// Mitsubishi GX Works2 project: PLC_GROUP_1   PLC: FX3G

// global labels: Global1
VAR_GLOBAL
  Start_day AT X007 : BOOL;
  Emergency_button AT X005 : BOOL;
  Inventory_check_flag AT M12 : BOOL;
  Day_activation_flag AT M0 : BOOL;
  Active_day AT Y007 : BOOL;
  Valid_inventory_flag AT M10 : BOOL;
  Start_making_flag AT M11 : BOOL;
  Special_gumigum_making AT M2 : BOOL;
  Regular_gumigum_making AT M1 : BOOL;
  Inventory_check AT X001 : BOOL;
  Petel_invetory AT D1200 : INT;
  Lemon_invetory AT D1202 : INT;
  Staiblaizer_invetory AT D1204 : INT;
  Gummy_bear_invetory AT D1206 : INT;
  Lemon AT D1112 : INT;
  Staibliazer AT D1114 : INT;
  Gummy_bear AT D1116 : INT;
  Analog_input AT D8280 : INT;
  IC_making_timer AT TC0 : BOOL;
  IC_making_timer_aprv AT TS0 : BOOL;
  Freezing_Timer AT TC1 : BOOL;
  Freezing_Timer_Aprv AT TS1 : BOOL;
  Regular_gumigum_mixing AT TC2 : BOOL;
  Regular_gumigum_mixing_apv AT TS2 : BOOL;
  Special_gumigum_mixing AT TC3 : BOOL;
  Special_gumigum_mixing_apv AT TS3 : BOOL;
  Flashlight_timer1 AT TC4 : BOOL;
  Flashlight_timer1_apv AT TS4 : BOOL;
  Flashlight_timer2 AT TC5 : BOOL;
  Flashlight_timer2_apv AT TS5 : BOOL;
  Start_mixing AT M13 : BOOL;
END_VAR
VAR_GLOBAL CONSTANT
  Constant2000 : INT := 2000;
  Constant2400 : INT := 2400;
  Req_petel_reg : INT := 280;
  Req_lemon_reg : INT := 455;
  Req_staibelaizer_reg : INT := 105;
  Req_gummybear_reg : INT := 28;
  Req_petel_spec : INT := 385;
  Req_lemon_spec : INT := 665;
  Req_staibelaizer_spec : INT := 210;
  Req_gummybear_spec : INT := 70;
END_VAR
VAR_GLOBAL
  Petel AT D1110 : INT;
END_VAR
VAR_GLOBAL CONSTANT
  timer50 : INT := 50;
END_VAR
VAR_GLOBAL
  timerTc2 AT TC2 : BOOL;
  IC_making AT Y000 : BOOL;
  Freezing_button AT X002 : BOOL;
  Freezing_lamp AT Y002 : BOOL;
END_VAR
VAR_GLOBAL CONSTANT
  timer30 : INT := 30;
END_VAR
VAR_GLOBAL
  Invalid_analog_input AT M14 : BOOL;
END_VAR
VAR_GLOBAL CONSTANT
  Regular_petel_container : INT := 350;
  Regular_lemon_container : INT := 490;
  Special_petel_container : INT := 560;
  Special_lemon_container : INT := 700;
END_VAR
VAR_GLOBAL
  Container_petel_IC AT D1130 : INT;
  Container_lemon_IC AT D1132 : INT;
  Petel_freezing_container AT D1140 : INT;
  Lemon_freezing_container AT D1142 : INT;
  Start_Freezing_Flag AT M15 : BOOL;
END_VAR
VAR_GLOBAL CONSTANT
  timer80 : INT := 80;
END_VAR
VAR_GLOBAL
  Temp_Sensor AT X003 : BOOL;
  Mixing_petel_container AT D1150 : INT;
  Mixing_lemon_container AT D1152 : INT;
  Flashlight_flag AT M16 : BOOL;
END_VAR
VAR_GLOBAL CONSTANT
  timer5 : INT := 5;
END_VAR
VAR_GLOBAL
  Flashlight1 AT Y005 : BOOL;
  Flashlight2 AT Y006 : BOOL;
  Packeges_counter AT D1160 : INT;
END_VAR
VAR_GLOBAL CONSTANT
  add1 : INT := 40;
END_VAR
VAR_GLOBAL
  Iteration_setting AT M30 : BOOL;
END_VAR
VAR_GLOBAL CONSTANT
  setting : INT;
END_VAR
VAR_GLOBAL
  Valid_p AT M40 : BOOL;
  Valid_l AT M41 : BOOL;
  Valid_s AT M42 : BOOL;
  Valid_g AT M43 : BOOL;
  check1 AT M50 : BOOL;
  check2 AT M51 : BOOL;
END_VAR
VAR_GLOBAL CONSTANT
  regular_gum : INT := 28;
  special_gum : INT := 70;
END_VAR
VAR_GLOBAL
  check3 AT M52 : BOOL;
  check4 AT M53 : BOOL;
  Analog_Output AT D8282 : INT;
END_VAR

// task Task_01 (event TRUE, interval 0, priority 31): POU_01

PROGRAM POU_01
(* structured ladder/FBD written out as ST: instructions are called as NAME(EN, inputs, outputs); _pN, _eN, _tN stand for wires *)
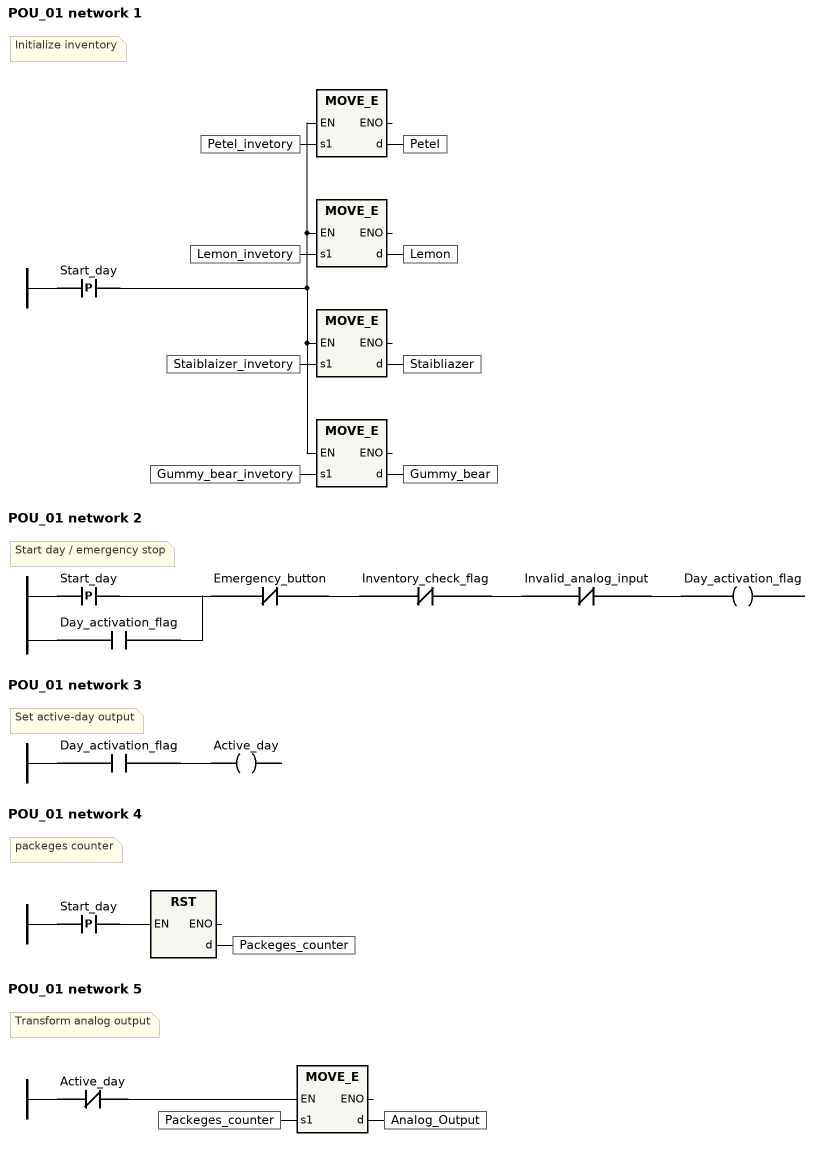
(* network 1 *)
(* Initialize inventory *)
_p1 := LDP(TRUE, Start_day);
MOVE_E(_p1, Petel_invetory, Petel);
MOVE_E(_p1, Lemon_invetory, Lemon);
MOVE_E(_p1, Staiblaizer_invetory, Staibliazer);
MOVE_E(_p1, Gummy_bear_invetory, Gummy_bear);
(* network 2 *)
(* Start day / emergency stop *)
Day_activation_flag := (((LDP(TRUE, Start_day) OR Day_activation_flag) AND NOT Emergency_button) AND NOT Inventory_check_flag) AND NOT Invalid_analog_input;
(* network 3 *)
(* Set active-day output *)
Active_day := Day_activation_flag;
(* network 4 *)
(* packeges counter *)
RST(LDP(TRUE, Start_day), Packeges_counter);
(* network 5 *)
(* Transform analog output *)
MOVE_E(NOT Active_day, Packeges_counter, Analog_Output);
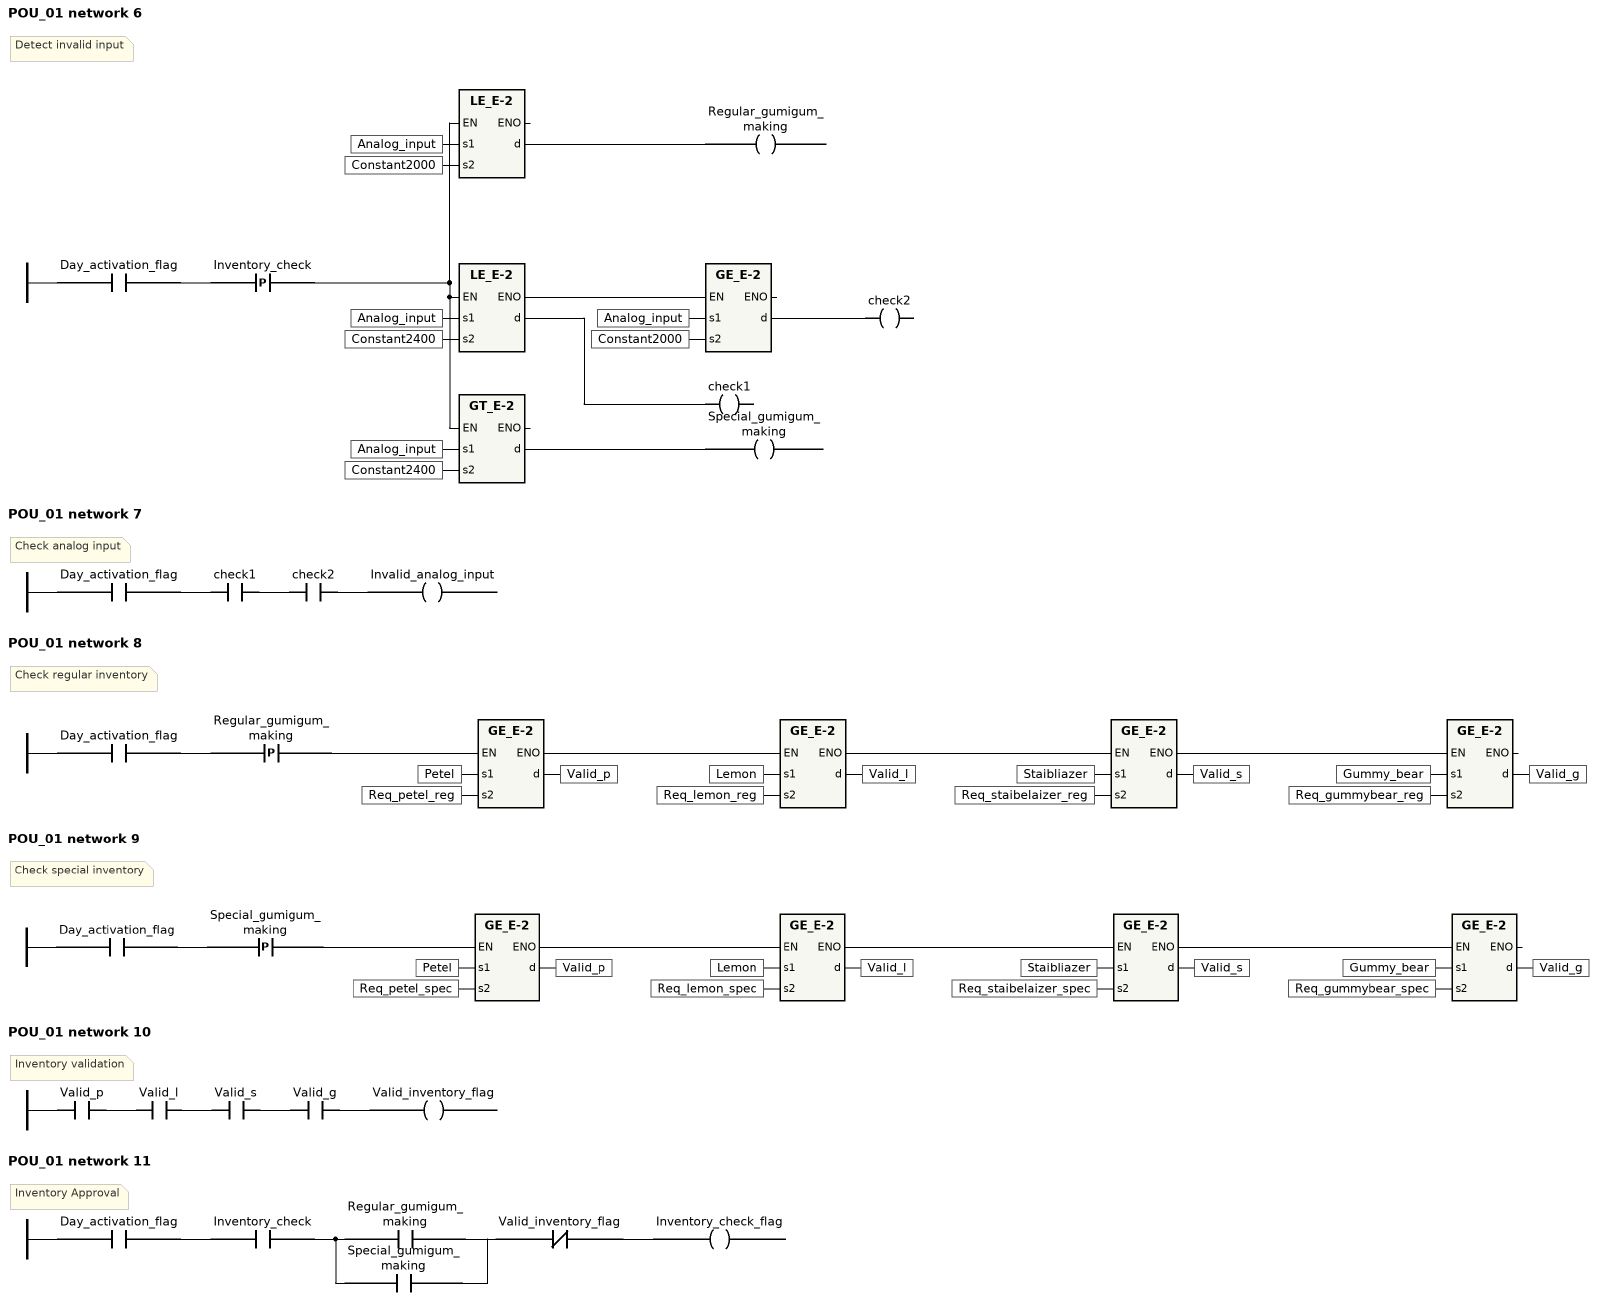
(* network 6 *)
(* Detect invalid input *)
_p1 := Day_activation_flag AND LDP(TRUE, Inventory_check);
LE_E(_p1, Analog_input, Constant2000, _t2);
Regular_gumigum_making := _t2;
GT_E(_p1, Analog_input, Constant2400, _t3);
Special_gumigum_making := _t3;
_e5 := LE_E(_p1, Analog_input, Constant2400, _t4);
GE_E(_e5, Analog_input, Constant2000, _t6);
check2 := _t6;
check1 := _t4;
(* network 7 *)
(* Check analog input *)
Invalid_analog_input := Day_activation_flag AND check1 AND check2;
(* network 8 *)
(* Check regular inventory *)
_e1 := GE_E(Day_activation_flag AND LDP(TRUE, Regular_gumigum_making), Petel, Req_petel_reg, Valid_p);
_e2 := GE_E(_e1, Lemon, Req_lemon_reg, Valid_l);
_e3 := GE_E(_e2, Staibliazer, Req_staibelaizer_reg, Valid_s);
GE_E(_e3, Gummy_bear, Req_gummybear_reg, Valid_g);
(* network 9 *)
(* Check special inventory *)
_e1 := GE_E(Day_activation_flag AND LDP(TRUE, Special_gumigum_making), Petel, Req_petel_spec, Valid_p);
_e2 := GE_E(_e1, Lemon, Req_lemon_spec, Valid_l);
_e3 := GE_E(_e2, Staibliazer, Req_staibelaizer_spec, Valid_s);
GE_E(_e3, Gummy_bear, Req_gummybear_spec, Valid_g);
(* network 10 *)
(* Inventory validation *)
Valid_inventory_flag := Valid_p AND Valid_l AND Valid_s AND Valid_g;
(* network 11 *)
(* Inventory Approval *)
_p1 := Day_activation_flag AND Inventory_check;
Inventory_check_flag := ((_p1 AND Regular_gumigum_making) OR (_p1 AND Special_gumigum_making)) AND NOT Valid_inventory_flag;
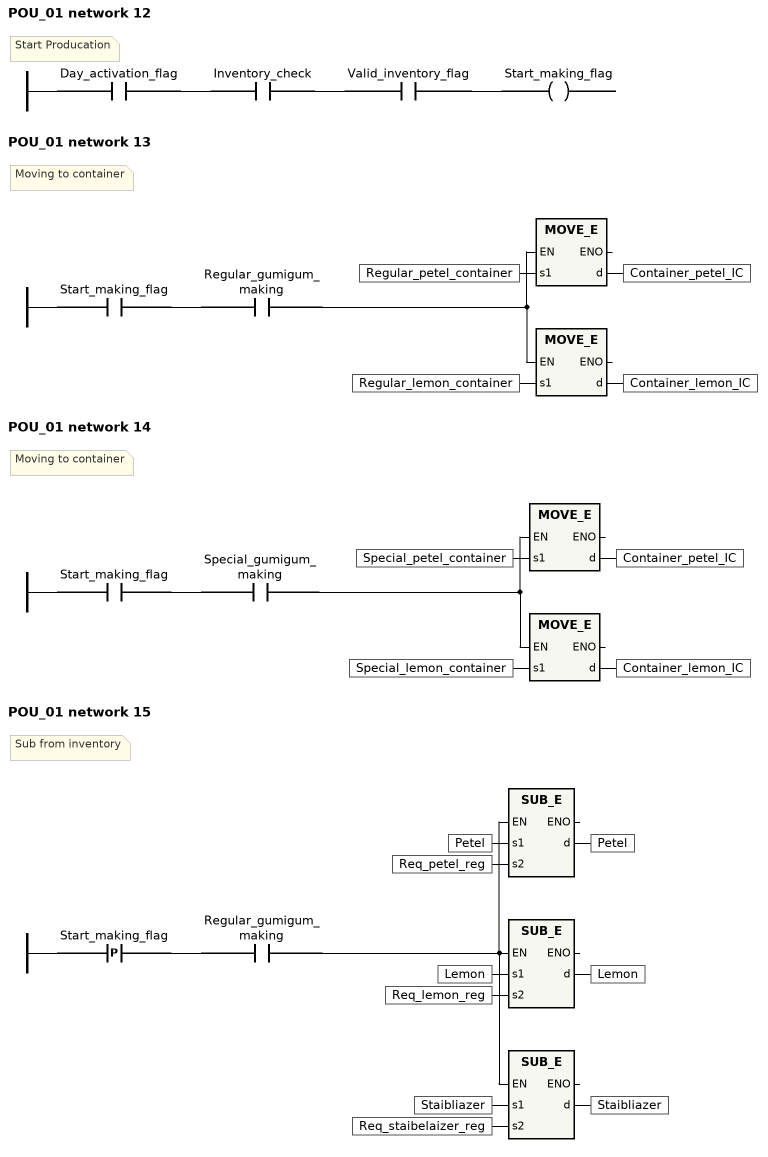
(* network 12 *)
(* Start Producation *)
Start_making_flag := Day_activation_flag AND Inventory_check AND Valid_inventory_flag;
(* network 13 *)
(* Moving to container *)
_p1 := Start_making_flag AND Regular_gumigum_making;
MOVE_E(_p1, Regular_petel_container, Container_petel_IC);
MOVE_E(_p1, Regular_lemon_container, Container_lemon_IC);
(* network 14 *)
(* Moving to container *)
_p1 := Start_making_flag AND Special_gumigum_making;
MOVE_E(_p1, Special_petel_container, Container_petel_IC);
MOVE_E(_p1, Special_lemon_container, Container_lemon_IC);
(* network 15 *)
(* Sub from inventory *)
_p1 := LDP(TRUE, Start_making_flag) AND Regular_gumigum_making;
SUB_E(_p1, Petel, Req_petel_reg, Petel);
SUB_E(_p1, Lemon, Req_lemon_reg, Lemon);
SUB_E(_p1, Staibliazer, Req_staibelaizer_reg, Staibliazer);
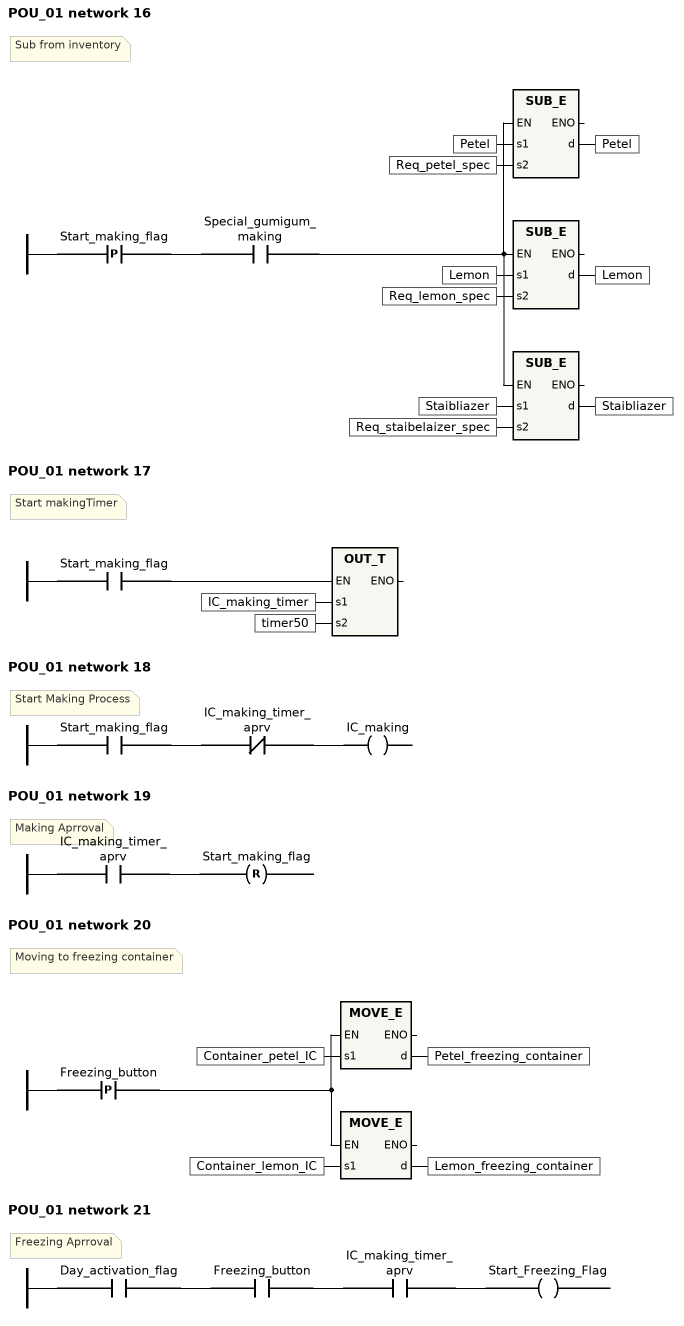
(* network 16 *)
(* Sub from inventory *)
_p1 := LDP(TRUE, Start_making_flag) AND Special_gumigum_making;
SUB_E(_p1, Petel, Req_petel_spec, Petel);
SUB_E(_p1, Lemon, Req_lemon_spec, Lemon);
SUB_E(_p1, Staibliazer, Req_staibelaizer_spec, Staibliazer);
(* network 17 *)
(* Start makingTimer *)
OUT_T(Start_making_flag, IC_making_timer, timer50);
(* network 18 *)
(* Start Making Process *)
IC_making := Start_making_flag AND NOT IC_making_timer_aprv;
(* network 19 *)
(* Making Aprroval *)
RST(IC_making_timer_aprv, Start_making_flag);
(* network 20 *)
(* Moving to freezing container *)
_p1 := LDP(TRUE, Freezing_button);
MOVE_E(_p1, Container_petel_IC, Petel_freezing_container);
MOVE_E(_p1, Container_lemon_IC, Lemon_freezing_container);
(* network 21 *)
(* Freezing Aprroval *)
Start_Freezing_Flag := Day_activation_flag AND Freezing_button AND IC_making_timer_aprv;
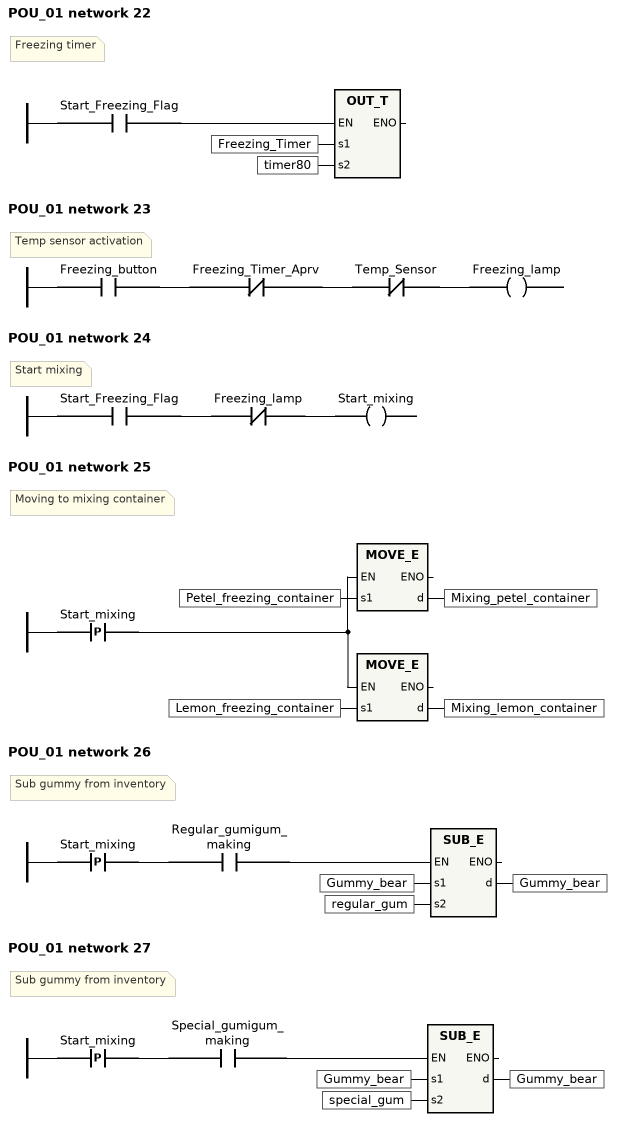
(* network 22 *)
(* Freezing timer *)
OUT_T(Start_Freezing_Flag, Freezing_Timer, timer80);
(* network 23 *)
(* Temp sensor activation *)
Freezing_lamp := Freezing_button AND NOT Freezing_Timer_Aprv AND NOT Temp_Sensor;
(* network 24 *)
(* Start mixing *)
Start_mixing := Start_Freezing_Flag AND NOT Freezing_lamp;
(* network 25 *)
(* Moving to mixing container *)
_p1 := LDP(TRUE, Start_mixing);
MOVE_E(_p1, Petel_freezing_container, Mixing_petel_container);
MOVE_E(_p1, Lemon_freezing_container, Mixing_lemon_container);
(* network 26 *)
(* Sub gummy from inventory *)
SUB_E(LDP(TRUE, Start_mixing) AND Regular_gumigum_making, Gummy_bear, regular_gum, Gummy_bear);
(* network 27 *)
(* Sub gummy from inventory *)
SUB_E(LDP(TRUE, Start_mixing) AND Special_gumigum_making, Gummy_bear, special_gum, Gummy_bear);
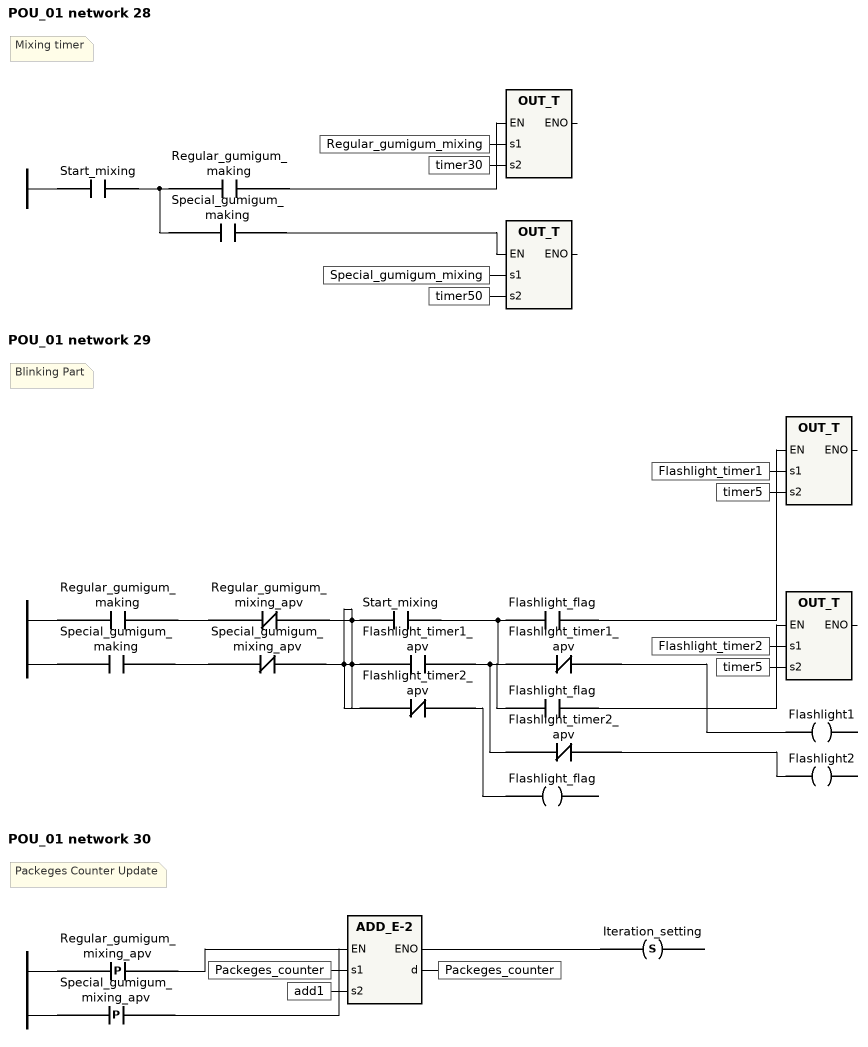
(* network 28 *)
(* Mixing timer *)
OUT_T(Start_mixing AND Regular_gumigum_making, Regular_gumigum_mixing, timer30);
OUT_T(Start_mixing AND Special_gumigum_making, Special_gumigum_mixing, timer50);
(* network 29 *)
(* Blinking Part *)
_p1 := (Regular_gumigum_making AND NOT Regular_gumigum_mixing_apv) OR (Special_gumigum_making AND NOT Special_gumigum_mixing_apv);
_p2 := _p1 AND Start_mixing;
OUT_T(_p2 AND Flashlight_flag, Flashlight_timer1, timer5);
Flashlight1 := _p2 AND NOT Flashlight_timer1_apv;
_p3 := _p1 AND Flashlight_timer1_apv;
OUT_T(_p3 AND Flashlight_flag, Flashlight_timer2, timer5);
Flashlight2 := _p3 AND NOT Flashlight_timer2_apv;
Flashlight_flag := _p1 AND NOT Flashlight_timer2_apv;
(* network 30 *)
(* Packeges Counter Update *)
_e1 := ADD_E(LDP(TRUE, Regular_gumigum_mixing_apv) OR LDP(TRUE, Special_gumigum_mixing_apv), Packeges_counter, add1, Packeges_counter);
SET(_e1, Iteration_setting);
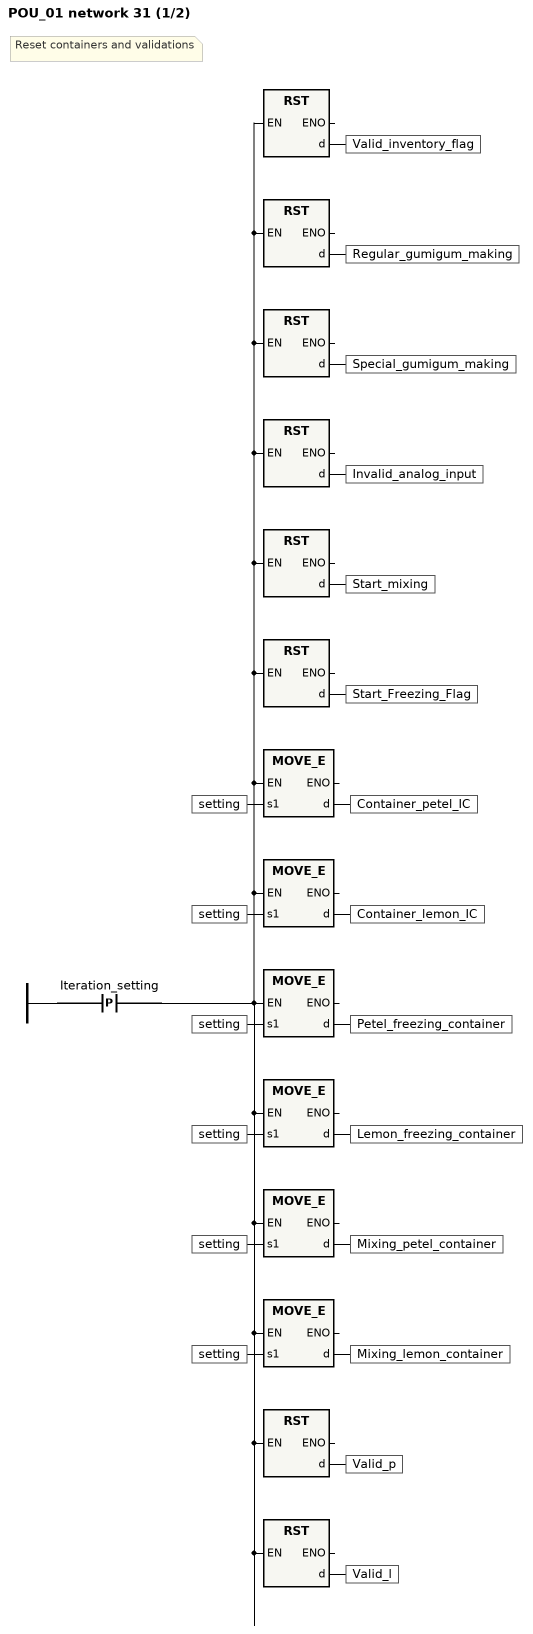
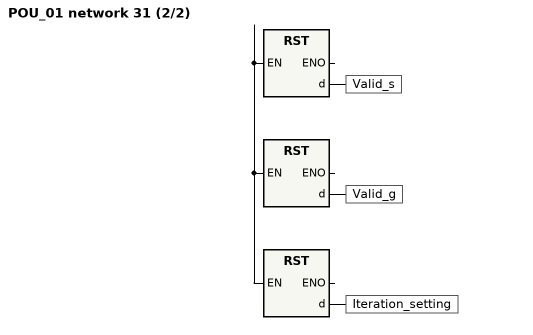
(* network 31 *)
(* Reset containers and validations *)
_p1 := LDP(TRUE, Iteration_setting);
RST(_p1, Valid_inventory_flag);
RST(_p1, Regular_gumigum_making);
RST(_p1, Special_gumigum_making);
RST(_p1, Invalid_analog_input);
RST(_p1, Start_mixing);
RST(_p1, Start_Freezing_Flag);
MOVE_E(_p1, setting, Container_petel_IC);
MOVE_E(_p1, setting, Container_lemon_IC);
MOVE_E(_p1, setting, Petel_freezing_container);
MOVE_E(_p1, setting, Lemon_freezing_container);
MOVE_E(_p1, setting, Mixing_petel_container);
MOVE_E(_p1, setting, Mixing_lemon_container);
RST(_p1, Valid_p);
RST(_p1, Valid_l);
RST(_p1, Valid_s);
RST(_p1, Valid_g);
RST(_p1, Iteration_setting);
END_PROGRAM
